# EPICS substitutions: pvNotepadApp/Db/longout_1.substitutions
#Substitution file for single record
file longout.template
{
     pattern { RECORD           }
             { $(HUTCH):NOTE:LONG:01 }
}
